{attribute addProperty BoxType "EK1122-0000-0018"}
{attribute addProperty Id "Beckhoff_ELXxxxxsub_EK1100EK1100_179A0949162"}
{attribute addProperty CRC "3457636952"}
{attribute addProperty SizeInBites "16"}
{attribute addProperty SizeInBytes "2"}
TYPE Beckhoff_ELXxxxxEK1122_CE175A58 EXTENDS EK1122_179A0949 :
STRUCT
	{attribute addProperty Name "Beckhoff_ELXxxxxsub_EK1100"}
	Beckhoff_ELXxxxxsub_EK1100 : EK1100_179A0949;
END_STRUCT
END_TYPE

(* stored: Version 1.2.0.0, ProductVersion 3.1.4024.9
   DUT Beckhoff_ELXxxxxEK1122_CE175A58: Id {c683a897-910b-4dfa-acf6-9698ed9fddf9} *)
